INTERFACE I_Timestamp

METHOD PUBLIC IsDurationElapsed : BOOL
VAR_INPUT
	Duration : TIME;
END_VAR
END_METHOD

END_INTERFACE

(* stored: Version 1.1.0.1, ProductVersion 3.1.4024.12
   Itf I_Timestamp: Id {d06ae25b-e200-418c-b777-6cb1fb5ec5c1}
   Method IsDurationElapsed: Id {e212337e-c991-4be9-96f7-7c2aa1c06dcf} *)
